{attribute 'GeneratedUsingTerminal: EL9227-4433-0018'}
{attribute addProperty BoxType "EL9227-4433-0018"}
{attribute addProperty Id "OCP_Inputs_Channel_1AT %I*OCP_Inputs_Channel_794A321B28OCP_Inputs_Channel_2AT %I*OCP_Inputs_Channel_794A321B28OCP_Outputs_Channel_1AT %Q*OCP_Outputs_Channel_010149342OCP_Outputs_Channel_2AT %Q*OCP_Outputs_Channel_010149342WcStateAT %I*WcState_9091E0EB2InfoDataAT %I*InfoData_32EB74EA10"}
{attribute addProperty CRC "1591982621"}
{attribute addProperty Size "72"}
TYPE EL9227_5EE3BA1D EXTENDS EtcSlaveTerminalBase_947E5A46 :
STRUCT
	{attribute addProperty Name "OCP_Inputs_Channel_1"}
	OCP_Inputs_Channel_1 : OCP_Inputs_Channel_794A321B;
	{attribute addProperty Name "OCP_Inputs_Channel_2"}
	OCP_Inputs_Channel_2 : OCP_Inputs_Channel_794A321B;
	{attribute addProperty Name "OCP_Outputs_Channel_1"}
	OCP_Outputs_Channel_1 : OCP_Outputs_Channel_01014934;
	{attribute addProperty Name "OCP_Outputs_Channel_2"}
	OCP_Outputs_Channel_2 : OCP_Outputs_Channel_01014934;
	{attribute addProperty Name "WcState"}
	WcState : WcState_9091E0EB;
	{attribute addProperty Name "InfoData"}
	InfoData : InfoData_32EB74EA;
END_STRUCT
END_TYPE

(* stored: Version 1.2.0.0, ProductVersion 3.1.4024.9
   DUT EL9227_5EE3BA1D: Id {8995d689-74ae-47ed-a17d-4dde4a3910a9} *)
